// TIA Portal V17 export
// export: Created 2026-04-13T11:12:45.0261807Z, ExportSetting WithDefaults, DisplayName Totally Integrated Automation Portal, DisplayVersion V17 Update 4, DisplayName TIA Portal Openness, DisplayVersion V17 Update 4, DisplayName TIA Portal Version Control Interface, DisplayVersion V17, DisplayName SINAMICS Startdrive Advanced, DisplayVersion V17, DisplayName SINAMICS Startdrive G130, G150, S120, S150, SINAMICS MV, S210, DisplayVersion V17, DisplayName SINAMICS Startdrive G110M, G120, G120C, G120D, G120P, G115D, DisplayVersion V17, DisplayName STEP 7 Professional, DisplayVersion V17 Update 4, DisplayName STEP 7 Safety, DisplayVersion V17, DisplayName WinCC Professional, DisplayVersion V17 Update 4
VAR_GLOBAL   // PLC tag table "默认变量表"
   System_Byte AT %MB1 : Byte;
   FirstScan AT %M1.0 : Bool;
   DiagStatusUpdate AT %M1.1 : Bool;
   AlwaysTRUE AT %M1.2 : Bool;
   AlwaysFALSE AT %M1.3 : Bool;
   Clock_Byte AT %MB0 : Byte;
   Clock_10Hz AT %M0.0 : Bool;
   Clock_5Hz AT %M0.1 : Bool;
   "Clock_2.5Hz" AT %M0.2 : Bool;
   Clock_2Hz AT %M0.3 : Bool;
   "Clock_1.25Hz" AT %M0.4 : Bool;
   Clock_1Hz AT %M0.5 : Bool;
   "Clock_0.625Hz" AT %M0.6 : Bool;
   "Clock_0.5Hz" AT %M0.7 : Bool;
   Tag_1 AT %MD800 : Real;
   Tag_2 AT %M810.0 : Bool;
   Tag_3 AT %MD820 : Real;
   Tag_4 AT %MD830 : Real;
   Tag_5 AT %MW840 : Int;
   Tag_6 AT %MD600 : DWord;
   Tag_7 AT %MD610 : DWord;
   Tag_8 AT %MD620 : DWord;
   Tag_9 AT %MD530 : DWord;
   Tag_10 AT %MD840 : DWord;
   Tag_12 AT %M100.0 : Bool;
   Tag_13 AT %M100.1 : Bool;
   自动运行报警 AT %M844.0 : Bool;
   自动停止 AT %M844.1 : Bool;
   Tag_14 AT %M110.0 : Bool;
   Tag_15 AT %M110.1 : Bool;
   Tag_16 AT %M111.0 : Bool;
   Tag_17 AT %M111.1 : Bool;
   M_手动修改 AT %M2000.0 : Bool;
   M_手动设定值 AT %MD2004 : Real;
   Tag_11 AT %MW300 : Word;
   Tag_18 AT %MW320 : Word;
   MQX清洗模式 AT %MW322 : Int;
   QQX清洗模式状态 AT %MW324 : Int;
   TEST AT %M111.2 : Bool;
END_VAR
